(*
SPDX-FileCopyrightText: © 2026 Oleksandr Tiutyk <trofimich@gmail.com>
SPDX-License-Identifier: MIT
License: https://opensource.org/license/mit
*)

(*!
<summary>
Demonstrates permission-controlled selection of traffic-light outputs. TrySetLight reports rejection or
exceptions without propagating them.
</summary>
*)

FUNCTION_BLOCK TrafficLight EXTENDS TOF_Automation.CompositeAutomationComponent<3> IMPLEMENTS ITrafficLight
VAR_STAT
	//! <summary>Class name shared by all instances of this function block.</summary>
	{attribute 'hide'} 
	_ClassName : STRING := __POUNAME();
END_VAR
VAR
	_RedLight : TOF_Devices_IO.DigitalOutput("RedLight", THIS^);
	_YellowLight : TOF_Devices_IO.DigitalOutput("YellowLight", THIS^);
	_GreenLight : TOF_Devices_IO.DigitalOutput("GreenLight", THIS^);
	
	_Children : ARRAY [0.._ChildCount - 1] OF TOF_Automation.IChildAutomationComponent := 
	[
		_RedLight, 
		_YellowLight, 
		_GreenLight
	];
END_VAR

{attribute 'monitoring' := 'call'}
PROPERTY FINAL ActiveLight : TRAFFIC_LIGHT_COLOR
GET
IF _RedLight.Value THEN
	ActiveLight := TRAFFIC_LIGHT_COLOR.RED;
ELSIF _YellowLight.Value THEN
	ActiveLight := TRAFFIC_LIGHT_COLOR.YELLOW;
ELSIF _GreenLight.Value THEN
	ActiveLight := TRAFFIC_LIGHT_COLOR.GREEN;
ELSE
	ActiveLight := TRAFFIC_LIGHT_COLOR.NO_COLOR;
END_IF
END_GET
END_PROPERTY

METHOD BindToIO
VAR_INPUT
	redLightRawValue : REFERENCE TO BOOL;
	yellowLightRawValue : REFERENCE TO BOOL;
	greenLightRawValue : REFERENCE TO BOOL;
END_VAR
_RedLight.BindToIO(rawValue := redLightRawValue);
_YellowLight.BindToIO(rawValue := yellowLightRawValue);
_GreenLight.BindToIO(rawValue := greenLightRawValue);
END_METHOD

{attribute 'monitoring' := 'call'}
PROPERTY FINAL BoundToIO : BOOL
GET
BoundToIO := _RedLight.BoundToIO AND_THEN _YellowLight.BoundToIO AND_THEN _GreenLight.BoundToIO;
END_GET
END_PROPERTY

{attribute 'monitoring' := 'call'}
PROPERTY FINAL Children : REFERENCE TO ARRAY [0.._ChildCount - 1] OF TOF_Automation.IChildAutomationComponent
GET
Children REF= _Children;
END_GET
END_PROPERTY

{attribute 'monitoring' := 'call'}
PROPERTY ClassName : REFERENCE TO STRING
GET
ClassName REF= _ClassName;
END_GET
END_PROPERTY

{attribute 'monitoring' := 'call'}
PROPERTY FINAL GreenLight : TOF_Devices_IO.IReadOnlyDigitalOutput
GET
GreenLight := _GreenLight;
END_GET
END_PROPERTY

{attribute 'monitoring' := 'call'}
PROPERTY NamespaceName : REFERENCE TO STRING
GET
NamespaceName REF= CurrentNamespace.Name;
END_GET
END_PROPERTY

{attribute 'monitoring' := 'call'}
PROPERTY FINAL RedLight : TOF_Devices_IO.IReadOnlyDigitalOutput
GET
RedLight := _RedLight;
END_GET
END_PROPERTY

{attribute 'monitoring' := 'call'}
PROPERTY SelfSize : ULINT
GET
SelfSize := XSIZEOF(THIS^);
END_GET
END_PROPERTY

(*!
<summary>Requests permission and attempts to select the traffic-light outputs.</summary>
<description>
Returns FALSE on rejection or a caught exception. Exceptions do not escape to the caller. Already changed
outputs are not rolled back; FALSE is not proof that all outputs are unchanged. A caught exception sets a
fixed rejection reason without allocating diagnostic objects. Fatal allocation observations return FALSE
before output changes after the permission callback. Earlier effects remain; the latch is preserved.
</description>
*)
METHOD TrySetLight : BOOL
VAR_INPUT
	color : TRAFFIC_LIGHT_COLOR;
END_VAR
VAR_IN_OUT
	rejectReason : WSTRING(255);
END_VAR
VAR
	actionDescriptor : TrySetLightActionDescriptor;
END_VAR
__TRY
	IF TOF_Core.DynamicMemoryManager.HasAllocationFailed THEN
		rejectReason := "Fatal allocation failure.";
		RETURN;
	END_IF

	// not usefull, only for demo how action permission checking can be implemented
	actionDescriptor.NewColor := color;

	IF NOT (TrySetLight := Parent.RequestActionPermission(
		actionDescriptor := actionDescriptor,
		requestingObject := THIS^,
		rejectReason := rejectReason
	))
	THEN
		RETURN;
	END_IF

	IF TOF_Core.DynamicMemoryManager.HasAllocationFailed THEN
		TrySetLight := FALSE;
		rejectReason := "Fatal allocation failure.";
		RETURN;
	END_IF

	_RedLight.Value := color = TRAFFIC_LIGHT_COLOR.RED;
	_YellowLight.Value := color = TRAFFIC_LIGHT_COLOR.YELLOW;
	_GreenLight.Value := color = TRAFFIC_LIGHT_COLOR.GREEN;
__CATCH
	TrySetLight := FALSE;
	rejectReason := "Unable to set traffic light.";
__ENDTRY

IF TOF_Core.DynamicMemoryManager.HasAllocationFailed THEN
	TrySetLight := FALSE;
	rejectReason := "Fatal allocation failure.";
END_IF
END_METHOD

{attribute 'monitoring' := 'call'}
PROPERTY FINAL YellowLight : TOF_Devices_IO.IReadOnlyDigitalOutput
GET
YellowLight := _YellowLight;
END_GET
END_PROPERTY

END_FUNCTION_BLOCK

(* stored: Version 1.1.0.1
   POU TrafficLight: Id {4a48deea-1b31-43e8-87e2-aa154a1466e2}, SpecialFunc None
   Folder Commands: Id {b0dba99f-d917-44fb-a6b0-98fb87cbba8e}
   Folder Statuses: Id {34522821-a59c-4891-b369-27c0febd3df8}
   Folder SubDevices: Id {b9cebfe2-cfee-4bf7-bbc2-7a57f1537e3e}
   Property ActiveLight: Id {467c94e8-e0fd-49e7-b0d7-7d25804d0224}
   Get Get: Id {c58454a7-f8c1-48c5-b685-f5be3d42efd3}
   Method BindToIO: Id {55cb475d-9082-491a-a7db-c010249b1dee}
   Property BoundToIO: Id {59765228-75e5-4a28-a5ce-f29eb52a2c07}
   Get Get: Id {2a0ad00d-a286-4691-80b4-d1cec1c85bff}
   Property Children: Id {f369897c-e280-452d-8cb5-1840f5d03f53}
   Get Get: Id {30214aac-7417-44f4-912f-019af48f8ceb}
   Property ClassName: Id {57d4725e-1474-4661-8746-ce344608dbc4}
   Get Get: Id {bf033ab4-a042-404c-85bc-755e1b6f3d73}
   Property GreenLight: Id {41aab368-6ec4-43bc-94ec-a15073d2d703}
   Get Get: Id {c5088c1e-3d45-46c5-a0ad-9786465d0b74}
   Property NamespaceName: Id {4ef76813-685e-4906-ba01-6114c2c08566}
   Get Get: Id {03ffe5c5-1446-4400-87f1-63e337477d04}
   Property RedLight: Id {580807e5-080b-4f74-a687-94c28623812c}
   Get Get: Id {59480cea-e4ff-4bea-b46e-1e0832dcc556}
   Property SelfSize: Id {0854c0b6-08bb-4062-b879-abc7c2048c2f}
   Get Get: Id {be673c01-8bac-444a-bd16-fa3be540c5df}
   Method TrySetLight: Id {66ac2472-cd7a-4221-b0c7-b8380631be67}
   Property YellowLight: Id {9e82f91e-7e2d-431b-8772-e8632c6f1a1a}
   Get Get: Id {ff958042-1f53-4b56-abc2-474fccdaecaf} *)
